INTERFACE I_ListObject

METHOD M_Add : BOOL
VAR_INPUT
	Object: 	I_Object;
END_VAR
END_METHOD

METHOD M_Clear
END_METHOD

METHOD M_Find : DINT
VAR_INPUT
	Object: 	I_Object;
END_VAR
END_METHOD

METHOD M_Get : I_Object
VAR_INPUT
	Index: 	DINT;
END_VAR
END_METHOD

METHOD M_Index : DINT
VAR_INPUT
	Object: 	I_Object;
END_VAR
END_METHOD

METHOD M_Remove : BOOL
VAR_INPUT
	Object: 	I_Object;
END_VAR
END_METHOD

PROPERTY P_Length : DINT
GET
END_GET
END_PROPERTY

END_INTERFACE

(* stored: Version 1.1.0.1
   Itf I_ListObject: Id {ebcd47ff-1663-4128-9d16-e6ffa6317543}
   Method M_Add: Id {78c2dc4e-c059-0ee4-1d4e-6a3f41393df7}
   Method M_Clear: Id {1d816771-7da2-09ff-2318-6eb9ddc155f7}
   Method M_Find: Id {9664ac8e-a0b9-0c4a-2c05-31740cc2cdc9}
   Method M_Get: Id {69c7a09c-f8ba-07d1-3063-8e31f9cac43e}
   Method M_Index: Id {e23e94e7-e402-01cb-2e81-d199ad68a010}
   Method M_Remove: Id {07441ba8-075c-0fa5-0895-940b56f7439a}
   Property P_Length: Id {eca1815b-8a98-0fae-3613-d611134bfecd}
   Get Get: Id {4d7f7332-0a18-4953-8b9f-ec4f6220f18f} *)
